FUNCTION_BLOCK FB_ShippingHoming EXTENDS FB_ActionBasic
VAR_INPUT
	xExecute : BOOL;
	xAbort : BOOL;
    FanucRobot : REFERENCE TO FB_FanucRobot_Basic;
	Homed : REFERENCE TO BOOL;
END_VAR
VAR_OUTPUT
	xAborted : BOOL;
	iErrorID : INT;
	ErrorMsg : STRING;
	RobotResetCMD : BOOL;
END_VAR
VAR
	StateBehaviour 		 : CBML.ETrigA;
	uiShippingHomingStep : UINT;
	FanucRobotCheckTon 	 : TON;
	ResetRobotDelay 	 :TON;
	fbExecuteEdgeDetect  :FB_EdgeDetect;
END_VAR

THIS^.IBehaviourModel := StateBehaviour;
StateBehaviour(xExecute := xExecute,
    xDone => xDone,
    xBusy => xBusy,
    xError => xError,
    xAbort := xAbort OR fbExecuteEdgeDetect.xFallingEdge,
    xAborted => xAborted);

//Error Msg
iErrorID := StateBehaviour._model.iErrorID;
ErrorMsg := M_GetErrorMsg(xErrorID := iErrorID);
FanucRobotCheckTon(PT := T#60S);

//Make sure that C# turns off execute to shut down the service
fbExecuteEdgeDetect(xInput :=xExecute);

ResetRobotDelay(PT:=T#300MS);

METHOD CleanupAction
VAR_INPUT
    xAbortProposed : BOOL;
    iErrorIDProposed: INT;
END_VAR
VAR_OUTPUT
    xComplete : BOOL := TRUE;
    xAbort: BOOL := xAbortProposed;
 	iErrorID : INT := iErrorIDProposed;
END_VAR
RobotResetCMD := FALSE;
FanucRobotCheckTon.IN := FALSE;
uiShippingHomingStep := 0;
END_METHOD

METHOD CyclicAction
VAR_INPUT
    itfTimingController : CBML.ITimingController;
END_VAR
VAR_OUTPUT
    xComplete : BOOL := TRUE;
    iErrorID : INT := 0;
END_VAR
xComplete := FALSE;
CASE uiShippingHomingStep OF
	0:
		FanucRobotCheckTon.IN := TRUE;
		IF FanucRobot.Error THEN
			RobotResetCMD := TRUE;
			ResetRobotDelay.IN:=TRUE;
		ELSE
			uiShippingHomingStep := 500;
		END_IF
		IF ResetRobotDelay.Q THEN
			ResetRobotDelay.IN :=FALSE;
			uiShippingHomingStep := 500;
		END_IF
		
		
	500:
		RobotResetCMD := FALSE;
		FanucRobot.OpMode := E_FanucRobotOpMode.RSR02;
		IF FanucRobot.Error THEN
			RobotResetCMD := TRUE;		
		END_IF
		IF FanucRobot._RSR2_Completed THEN
			uiShippingHomingStep := 600;
		END_IF
	600:
		FanucRobot.OpMode := E_FanucRobotOpMode.RSR01;
		IF FanucRobot._RSR1_Ready THEN
			uiShippingHomingStep := 700;
		END_IF
	700:
		FanucRobotCheckTon.IN := FALSE;
		Homed := TRUE;
		xComplete := TRUE;
END_CASE

IF FanucRobotCheckTon.Q THEN
	iErrorID := 4;
END_IF
END_METHOD

METHOD ExitAction
VAR_INPUT
    xAfterCleanup : BOOL;
    xInCopyCode : BOOL;
END_VAR
END_METHOD

METHOD M_GetErrorMsg : T_MaxString
VAR_INPUT
	xErrorID: INT;
END_VAR

VAR
	
END_VAR
CASE xErrorID OF
    0:
        M_GetErrorMsg := 'No Error';
    1:
        M_GetErrorMsg := 'Action time out';
    2:
        M_GetErrorMsg := 'Cylinder not ready';
    3:
        M_GetErrorMsg := 'Motor not ready';
    4:
		M_GetErrorMsg := 'FanucRobot can not homing';
END_CASE
END_METHOD

METHOD ResetAction
VAR_OUTPUT
    xComplete : BOOL := TRUE;
END_VAR
FanucRobotCheckTon.IN := false;
END_METHOD

METHOD StartAction
VAR_OUTPUT
    xComplete : BOOL := TRUE;
	iErrorID : INT := 0;
END_VAR
Homed := FALSE;
FanucRobotCheckTon.IN := FALSE;
uiShippingHomingStep := 0;
END_METHOD

END_FUNCTION_BLOCK

(* stored: Version 1.1.0.1, ProductVersion 3.1.4024.13
   POU FB_ShippingHoming: Id {fb6a1860-c382-494a-99f6-2de10876296e}, SpecialFunc None
   Method CleanupAction: Id {f4a4a7bd-b035-4c68-8efe-6ad0c9c5f25b}
   Method CyclicAction: Id {ccbe0fb7-3c8a-435f-b091-6473cfa1a63d}
   Method ExitAction: Id {b40aaad3-b319-49ad-ab2a-b5db16cceaaa}
   Method M_GetErrorMsg: Id {03eac412-96d4-4e84-bf40-8d06670d8278}
   Method ResetAction: Id {a5d6e6fc-9b41-4dd3-92ef-8e0382f51f5a}
   Method StartAction: Id {a77f2f89-4696-4442-828d-0460ba5f894c} *)
